// TIA Portal V18 export
FUNCTION "AHURegsAndTargetStatesInComfortOpMode" : Void   // FC60033, LAD
{ S7_Optimized_Access := 'TRUE' }
VERSION : 0.1
// Operation Modes                                                 Unit State
// 0=                                                                            0=Stopped
// 1                                                                              1=Checking-up  
// 2                                                                              2=Preheating
// 3 = Comfort                                                           3=Starting 
//                                                                                 4=RecirculatingOperation (Protection)
//                                                                                 Not 5=Sustained Mode (Economy)
//                                                                                 Not 6=Sustained Mode (PreComfort setpoints) 
//                                                                                 7=Comfort  operation
//                                                                                 Not 8=Night Cooling
//                                                                                 9=Stopping
//                                                                                 10=Blocking
//                                                                                 11=FrostProtecting
// stored: AutoNumber false, IsIECCheckEnabled false, SetENOAutomatically false, UDAEnableTagReadback false
   VAR_INPUT
      iUnitID : Int;
      cActualOpMode : Byte;
      cHeatingRegCfg : Byte;
      cCoolingRegCfg : Byte;
      cIAQRegCfg : Byte;
      cBuildingdPRegCfg : Byte;
   END_VAR
   VAR_OUTPUT
      cTargetState : Byte;
      cHeatingRegState : Byte;
      cCoolingRegState : Byte;
      cIAQRegState : Byte;
      cBuildingdPRegState : Byte;
   END_VAR
BEGIN

REGION Network 1 (SCL)
   IF NOT "AHUAlarms".Summary.FrostAlarm[#iUnitID] AND NOT "AHUAlarms".Summary.BlockingAlarm[#iUnitID] THEN
       // Statement section IF
       #cTargetState := 7;
       #cHeatingRegState := #cHeatingRegCfg;
       #cCoolingRegState := #cCoolingRegCfg;
       #cIAQRegState := #cHeatingRegCfg;
       #cHeatingRegState := #cHeatingRegCfg;


   END_IF;
END_REGION
END_FUNCTION
